(* CODESYS project SECoP-PLC
   Author: Zeus Castillo
   Company: ILL
   DefaultNamespace: SECoP
   Description: Library for configuring a Codesys-based PLC as a SEC Node
   DocFormat: reStructuredText
   LanguageModelAttribute: qualified-access-only
   Placeholder: SECoP
   Title: SECoP
   Version: 1.1.0.0

Project tree, tasks and I/O mapping:
  libraries: CAA Types Extern, 3.5.17.0 (CAA Technical Workgroup); CAA FB Factory, 3.5.19.0 (CAA Technical Workgroup); Common Behaviour Model, 4.0.0.0 (CODESYS); StringUtils, 3.5.20.0 (System); Util, 3.5.21.0 (System); Standard, 3.5.18.0 (System); SysMem, 3.5.17.0 (System); TcpUdpCommunication, 2.3.2.0 (Schneider Electric); JSON Utilities SL, 1.11.0.0 (CODESYS)
  global variables GCL
  global variables GPL
  global variables GVL
  data type ET_TimestampSource
  function block FB_SecNode [ST]: M_ReturnSecNodeError
  data type ST_SecNode
  data type ST_Timestamp
  program Server [ST]: A_MessageFragmentation, A_ParseClientMessage, A_ProcessClientRequest
  function GetLibVersion [ST]
  function GetLibVersionNumber [ST]
  function IsLibReleased [ST]
  data type ET_BaseClass
  data type ET_StatusCode
  function block FB_BaseModuleReadable [ST]: A_GenerateStatusDataReport, A_HandlePollintervalChange, A_ReturnErrorNoSuchCommand, A_ReturnErrorReadOnly, A_ReturnErrorWrongType, M_AddDataReportToReplyMessage, M_CheckIfDataIsNumeric, M_ExtractTargetLimitsFromTuple, M_GenerateTargetLimitsDataReport, M_JsonDecodeString, M_JsonEncodeString, M_ReturnRangeError
  data type ST_BaseModuleReadable
  data type ST_HandlePollinterval
  data type ST_ModuleStatus
  data type ST_Subscriber
  data type ST_TargetWrite
  data type ST_TargetDrive
  function block FB_diTargetDrive [ST]
  function block FB_IsStableNum [ST]
  function block FB_MonitorNumValue [ST]
  function block FB_MonitorSmallString [ST]
  function block FB_sTargetDrive [ST]
  global variables GPL_TcpServer_SE
*)

// ET_TimestampSource
{attribute 'qualified_only' := ''}
{attribute 'strict' := ''}
TYPE ET_TimestampSource :
(
	/// Value's timestamp to be obtained from the ECS (equipment that controls the hardware)
	Ecs := 1,
	/// Value's timestamp to be generated by this SEC node (this controller)				
	ThisSecNode := 2
);
END_TYPE

// ST_SecNode
TYPE ST_SecNode :
STRUCT
	// Firmware
	sFirmware: STRING := 'secnodeplc-1.0';
	// Protocol version
	sSecopVersion: STRING := 'V2019-09-16';	
	/// TCP server IP address
	sTcpServerIp: STRING(15);
	/// TCP server port
	uiTcpServerPort: UINT;
	// TCP server Eth interface link up
	xTcpServerInterfaceReady : BOOL:= FALSE;
	/// Default poll interval (to be used for modules that don´t have an independent pollinterval configured)
	timPollInterval: TIME := TIME#5S;
	/// Timestamp
	sTimestamp: STRING;
	/// Error report
	stErrorReport: ST_ErrorReport;
	// Module list
	asModule: ARRAY[1..GPL.Gc_uiMaxNoOfModules] OF STRING;
	// Action list
	asAction: ARRAY[1..GPL.Gc_uiMaxNoOfActions] OF STRING := ['*IDN?', 'describe', 'activate', 'deactivate', 'ping', 'read', 'change', 'do'];	
	// Structure report
	sStructureReport: STRING(GPL.Gc_uiMaxSizeMessage);
END_STRUCT
END_TYPE

// ST_Timestamp
TYPE ST_Timestamp :
STRUCT
	etSource: ET_TimestampSource;
	sValue: STRING;
END_STRUCT
END_TYPE

// ET_BaseClass
{attribute 'qualified_only' := ''}
{attribute 'strict' := ''}
TYPE ET_BaseClass : // Module's interface class 
(
	//Communicator := 0,
	Readable := 1,
	Writable := 2,
	Drivable := 3
);
END_TYPE

// ET_StatusCode
{attribute 'qualified_only' := ''}
{attribute 'strict' := ''}
TYPE ET_StatusCode : // Module's status code
(
	/// implemented
	Disabled := 0,
	Idle := 100,
	Warn := 200,
	Busy := 300,
	Error := 400,
	/// not implemented yet
	Persist := 101,
	Prepare := 301,
	Ramping := 302,
	Finish := 303
);
END_TYPE

// ST_BaseModuleReadable
TYPE ST_BaseModuleReadable :
STRUCT
	/// Interface class
	etInterfaceClass: ET_BaseClass;
	/// Name
	sName: STRING(80);
	/// Description
	sDescription: STRING(255);
	/// Current status of the module
	stStatus: ST_ModuleStatus;
	/// Polling interval of the module
	stPollInterval: ST_HandlePollinterval;
	/// Array of currently subscribed clients
	astSubscriberList: ARRAY[1..GPL.Gc_uiMaxNoOfClients] OF ST_Subscriber;
	/// Timestamp
	sTimestamp: STRING;
	/// Error report		
	stErrorReport: ST_ErrorReport;
END_STRUCT
END_TYPE

// ST_HandlePollinterval
TYPE ST_HandlePollinterval : // Module's poll intervall handling data
STRUCT
	lrValue: LREAL := 5.0;
	lrMin: LREAL := 0.5;
	lrMax: LREAL := 120.0;
	xReadOnly: BOOL := FALSE;
//	stPollintervalChangeClient: ST_Subscriber; // Client that sent the last pollinterval change request	
END_STRUCT
END_TYPE

// ST_ModuleStatus
TYPE ST_ModuleStatus : // Module's status data
STRUCT
	/// Staus code
	etCode: ET_StatusCode;
	/// Status description
	sDescription: STRING(GPL.Gc_uiMaxSizeDescription);
	/// Module inactive (flag) becomes unavailable for SECoP clients e.g. due to equipment configuration
	xInactive : BOOL; 
END_STRUCT
END_TYPE

// ST_Subscriber
TYPE ST_Subscriber : // Subscribed SECoP client data
STRUCT
	/// IP Address
	sIp: STRING(15);
	/// Assigned port number
	uiPort: UINT;
END_STRUCT
END_TYPE

// ST_TargetWrite
TYPE ST_TargetWrite : // Module's target change handling data
STRUCT
	/// Interlock
	xPossible: BOOL;
	/// Client that sent the last target change request	
	stTargetChangeClient: ST_Subscriber;
END_STRUCT
END_TYPE

// ST_TargetDrive
TYPE ST_TargetDrive : // Module's target drive handling data
STRUCT
	/// State machine. 0:Idle, 1:Request, 2:Applied in hardware, 3:Driving, 4:Completed
	uiState: UINT;
	/// Timeout to reach target
	timTimeout: TIME := TIME#10M0S0MS;
	/// Clients that sent a target change request while the target is still driving (module BUSY)
	astClientList: ARRAY[1..GPL.Gc_uiMaxNoOfClients] OF ST_Subscriber;
	/// Stay at current value command
	xStopCmd: BOOL;
	/// Client that sent the last stop command
	stStopCmdClient: ST_Subscriber;
END_STRUCT
END_TYPE

// GCL
{attribute 'qualified_only'}
VAR_GLOBAL CONSTANT
	Gc_uiMaxSizeIdentifier : UINT := 64; // Max. size of the specifier (e.g. module and accessible name) inside the message	
	Gc_uiMaxSizeAction : UINT := 64; // Max. size of action inside the message
	Gc_uiMaxSizeSpecifier : UINT := (GCL.Gc_uiMaxSizeIdentifier*2)+1; // Max. size of action inside the message
	Gc_uiMaxSizeClientMessage : UINT := Gc_uiMaxSizeAction+Gc_uiMaxSizeSpecifier+GPL.Gc_uiMaxSizeData+5; // Max. size of a messages received from SECoP clients	
	Gc_uiMaxNbOfSubmessages : UINT := 3; // Action, specier and data, separated by a white space character (\x20)
	Gc_dwLibVersionNumber : DWORD := 16777216; // Manual copy of GetLibVersionNumber(). Used in sec node app to create compile-time warning if > max.version supported by code generator
END_VAR

// GPL
{attribute 'qualified_only'}
{attribute 'parameterlist'}
VAR_GLOBAL CONSTANT
	Gc_uiMaxSizeMessage : UINT := 20000; // Max. size of a messages sent to SECoP clients
	Gc_uiMaxSizeData : UINT := 2000; // Max. size of the Data part of a SECoP message (a message = Action + Specifier (e.g. module:accessible) + Data)
	Gc_uiMaxSizeDescription : UINT := 500; // Max. size of the description in the Status or Error Report message 		
	Gc_uiMaxNoOfClients : UINT := 3; // Max. number of simultaneous connected clients
	Gc_uiMaxNoOfModules : UINT := 100; // Max. number of implemented modules in the SEC Node
	Gc_uiMaxNoOfActions : UINT := 15; // Max. number of implemented actions in the SEC Node
END_VAR

// GVL
{attribute 'qualified_only'}
VAR_GLOBAL
	G_st_SecNode : ST_SecNode; // SEC Node 
	G_ProcessModules : I_ProcessModules; // Process modules interface
	G_xProcessModulesAssigned : BOOL := FALSE; // (Flag) Process modules interface linked in application
	G_xJsonLibInstalled : BOOL := FALSE; // (Flag) JSON Utilities SL library installed in application (license required)
END_VAR

// GPL_TcpServer_SE
{attribute 'qualified_only'}
{attribute 'parameterlist'}
VAR_GLOBAL CONSTANT
	/// Max buffer size for sending/receiving data in one function call when using the Send/Receive methods from the TcpUdpCommunication library.
	/// M251: 2048. M262: 20000 for instance
	Gc_uiDataTransferChunkSize: UINT := 20000;
	/// Max. size of a message to be sent. If 'Gc_uiSendingMessageMaxSize' is greater than 'GVL_SaneTcp.Gc_uiDataTransferChunkSize', it will be split into several chunks that will be sent in consecutive function calls.
	/// For M262, it is recommended to be ser to same value as 'Gc_uiDataTransferChunkSize' to avoid splitting
	Gc_uiSendingMessageMaxSize: UINT := 20000;
END_VAR

// FB_SecNode
FUNCTION_BLOCK FB_SecNode
VAR_INPUT
	/// Action identifier (type of request: describe, activate...)
	i_sAction: STRING;
	/// Module name (empty for SEC node global actions which are not module-related)
	i_sModule: STRING(GCL.Gc_uiMaxSizeIdentifier);
	/// used as id for "ping" requests (the "pong" reply contains exactly the same id)	
	i_sArgument: STRING(((2 * GCL.Gc_uiMaxSizeIdentifier) + 1));
	/// Client sent a new request that needs processing
	i_xSyncModeRequest: BOOL;
	/// Action is implemented in this SEC node
	i_xActionIsImplemented: BOOL;
	/// Specifier format correct
	i_xSpecifierFormatOk: BOOL;
END_VAR
VAR_IN_OUT
	iq_stSecNode: ST_SecNode;
	/// Reply message
	iq_sReplyMessage: STRING(GPL.Gc_uiMaxSizeMessage);
END_VAR
VAR
	/// Flags
	iModuleIndex: INT;
END_VAR


// Process client request in sync mode
IF i_xSyncModeRequest THEN

	// Action not implemented
	IF NOT i_xActionIsImplemented THEN
		
		IF i_sAction='logging' OR i_sAction='check' THEN
			// Return "NotImplemented" error
			iq_stSecNode.stErrorReport.sClass := 'NotImplemented';
			iq_stSecNode.stErrorReport.sDescription := i_sAction;
			StrConcatA(pstFrom:= ADR(' is not implemented on this SEC node'), pstTo:= ADR(iq_stSecNode.stErrorReport.sDescription), iBufferSize:= UINT_TO_INT(GPL.Gc_uiMaxSizeDescription));
			M_ReturnSecNodeError(i_xErrorLatched:= FALSE);	
		
		ELSE // Return "ProtocolError" error
			iq_stSecNode.stErrorReport.sClass := 'ProtocolError';
			iq_stSecNode.stErrorReport.sDescription := 'Unknown action';
			M_ReturnSecNodeError(i_xErrorLatched:= FALSE);				
		END_IF

	// Specifier format error
	ELSIF NOT i_xSpecifierFormatOk THEN
		// Return "ProtocolError" error
		iq_stSecNode.stErrorReport.sClass := 'ProtocolError';
		iq_stSecNode.stErrorReport.sDescription := 'Specifier format error';
		M_ReturnSecNodeError(i_xErrorLatched:= FALSE);			
		
	ELSE
		
		// Process SEC Node request (global action which is not module-related)
		IF StrIsNullOrEmptyA(ADR(i_sModule)) = TRUE THEN
			// identification
				IF i_sAction = '*IDN?' THEN
					
					// Prepare reply message: ISSE,SECoP,(optional)<date indicating pre-release draft of the specin use>,< released version of SECoP>
					iq_sReplyMessage := 'ISSE,SECoP,2026-03-10,v2.0';
					M_AddTermToReplyMessage(i_etTerminator:= ET_Terminator.LineFeed); // Append line feed terminator to the message				
					
				// description
				ELSIF i_sAction = 'describe' THEN 
					
					// Prepare reply message: describing␣.␣<structure-report>
					iq_sReplyMessage := 'describing . ';
					StrConcatA(pstFrom:= ADR(iq_stSecNode.sStructureReport), pstTo:= ADR(iq_sReplyMessage), iBufferSize:= UINT_TO_INT(GPL.Gc_uiMaxSizeMessage));
					M_AddTermToReplyMessage(i_etTerminator:= ET_Terminator.LineFeed); // Append line feed terminator to the message	
				
				// activate updates
				ELSIF i_sAction = 'activate' THEN
		
					// Append action end message. Update messages were already inserted by the module FBs 			
					StrConcatA(pstFrom:= ADR('active'), pstTo:= ADR(iq_sReplyMessage), iBufferSize:= UINT_TO_INT(GPL.Gc_uiMaxSizeMessage));
					M_AddTermToReplyMessage(i_etTerminator:= ET_Terminator.LineFeed); // Append line feed terminator to the message				
	
				
				// deactivate updates
				ELSIF i_sAction = 'deactivate' THEN
					
					StrConcatA(pstFrom:= ADR('inactive'), pstTo:= ADR(iq_sReplyMessage), iBufferSize:= UINT_TO_INT(GPL.Gc_uiMaxSizeMessage));	
					M_AddTermToReplyMessage(i_etTerminator:= ET_Terminator.LineFeed); // Append line feed terminator to the message					
				
				// heartbeat. ping␣<identifier>
				ELSIF i_sAction = 'ping' THEN 
					
					// Prepare reply message: pong␣<identifier>␣<data-report>
					iq_sReplyMessage := 'pong ';
					StrConcatA(pstFrom:= ADR(i_sArgument), pstTo:= ADR(iq_sReplyMessage), iBufferSize:= UINT_TO_INT(GPL.Gc_uiMaxSizeMessage));
					StrConcatA(pstFrom:= ADR(' [null, {"t": '), pstTo:= ADR(iq_sReplyMessage), iBufferSize:= UINT_TO_INT(GPL.Gc_uiMaxSizeMessage));
					StrConcatA(pstFrom:= ADR(iq_stSecNode.sTimestamp), pstTo:= ADR(iq_sReplyMessage), iBufferSize:= UINT_TO_INT(GPL.Gc_uiMaxSizeMessage));
					StrConcatA(pstFrom:= ADR('}]'), pstTo:= ADR(iq_sReplyMessage), iBufferSize:= UINT_TO_INT(GPL.Gc_uiMaxSizeMessage));
					M_AddTermToReplyMessage(i_etTerminator:= ET_Terminator.LineFeed); // Append line feed terminator to the message
				END_IF
			
		ELSE // Check if the module specified on the client request is recognised. Return error otherwise
			FOR iModuleIndex := 1 TO UINT_TO_INT(GPL.Gc_uiMaxNoOfModules) BY 1 DO
				IF iq_stSecNode.asModule[iModuleIndex]=i_sModule THEN
					EXIT;
				END_IF
				IF StrIsNullOrEmptyA(ADR(iq_stSecNode.asModule[iModuleIndex])) THEN // end of module list reached
					// Return "NoSuchModule" error
					iq_stSecNode.stErrorReport.sClass := 'NoSuchModule';
					iq_stSecNode.stErrorReport.sDescription := i_sModule;
					StrConcatA(pstFrom:= ADR(' is not configured on this SEC node'), pstTo:= ADR(iq_stSecNode.stErrorReport.sDescription), iBufferSize:= UINT_TO_INT(GPL.Gc_uiMaxSizeDescription));
					M_ReturnSecNodeError(i_xErrorLatched:= FALSE);	
					EXIT;
				END_IF
			END_FOR				
		END_IF
	END_IF
END_IF

METHOD M_ReturnSecNodeError : BOOL
VAR_INPUT
	i_xErrorLatched: BOOL;
END_VAR

// Raise error flag
iq_stSecNode.stErrorReport.xActive := TRUE;	

// Build error report
StrConcatA(pstFrom:= ADR('error_'), pstTo:= ADR(iq_sReplyMessage), iBufferSize:= UINT_TO_INT(GPL.Gc_uiMaxSizeMessage));
StrConcatA(pstFrom:= ADR(i_sAction), pstTo:= ADR(iq_sReplyMessage), iBufferSize:= UINT_TO_INT(GPL.Gc_uiMaxSizeMessage));
StrConcatA(pstFrom:= ADR(' ["'), pstTo:= ADR(iq_sReplyMessage), iBufferSize:= UINT_TO_INT(GPL.Gc_uiMaxSizeMessage));	
StrConcatA(pstFrom:= ADR(iq_stSecNode.stErrorReport.sClass), pstTo:= ADR(iq_sReplyMessage), iBufferSize:= UINT_TO_INT(GPL.Gc_uiMaxSizeMessage));
StrConcatA(pstFrom:= ADR('","'), pstTo:= ADR(iq_sReplyMessage), iBufferSize:= UINT_TO_INT(GPL.Gc_uiMaxSizeMessage));
StrConcatA(pstFrom:= ADR(iq_stSecNode.stErrorReport.sDescription), pstTo:= ADR(iq_sReplyMessage), iBufferSize:= UINT_TO_INT(GPL.Gc_uiMaxSizeMessage));
StrConcatA(pstFrom:= ADR('",{"t":'), pstTo:= ADR(iq_sReplyMessage), iBufferSize:= UINT_TO_INT(GPL.Gc_uiMaxSizeMessage));
StrConcatA(pstFrom:= ADR(iq_stSecNode.sTimestamp), pstTo:= ADR(iq_sReplyMessage), iBufferSize:= UINT_TO_INT(GPL.Gc_uiMaxSizeMessage));
StrConcatA(pstFrom:= ADR('}]'), pstTo:= ADR(iq_sReplyMessage), iBufferSize:= UINT_TO_INT(GPL.Gc_uiMaxSizeMessage));	

// Append line feed terminator to the message
M_AddTermToReplyMessage(i_etTerminator:= ET_Terminator.LineFeed);	

// Unlatch error
IF NOT i_xErrorLatched THEN
	iq_stSecNode.stErrorReport.xActive := FALSE;
END_IF
END_METHOD

END_FUNCTION_BLOCK

// Server
PROGRAM Server // Sec node TCP server
VAR_INPUT
	xCmdClearResult: BOOL; /// Reset Cmd. Clear last diagnostic messages and alarms on rising edge
	xCmdDisconnectAll: BOOL; /// Disconnect all clients on rising edge	
	xCmdClose: BOOL; /// Stop listening (close port) on rising edge
END_VAR
VAR
{IF project_defined(SCHNEIDER_ELECTRIC)} 
	// SCHNEIDER_ELECTRIC Tcp Server handling
	fbTcpServer: FB_ASCIIoverTCPserver_SE;	
	fbReceivedData: ARRAY[1..TCPUDP.GPL.Gc_uiTCPServerMaxConnections] OF FB_MonitorNumValue;
	fbDisconnectedClientIp: ARRAY[1..TCPUDP.GPL.Gc_uiTCPServerMaxConnections] OF FB_MonitorSmallString;
	fbDisconnectedClientPort: ARRAY[1..TCPUDP.GPL.Gc_uiTCPServerMaxConnections] OF FB_MonitorNumValue;
	astClientInfo: ARRAY [1..TCPUDP.GPL.Gc_uiTCPServerMaxConnections] OF ST_ClientInfo_SE;
	asMessageToSend: ARRAY[1..TCPUDP.GPL.Gc_uiTCPServerMaxConnections] OF STRING(GPL_TcpServer_SE.Gc_uiSendingMessageMaxSize);
	sTcpServerState: STRING;
	sTcpServerResult: STRING;
	sLastErrorDiagMessage: STRING;
	uiNbOfConnectedClients: UINT;
	xPortOpen: BOOL;
	sDiagMessage: STRING;
	/// Auxiliary variables
	xMessageFragNeeded : BOOL := GPL_TcpServer_SE.Gc_uiDataTransferChunkSize < GPL_TcpServer_SE.Gc_uiSendingMessageMaxSize; // Message fragmentation needed	
	iStartPos: INT;
	iEndPos: INT;
	sDisconnectedCientIp: STRING;
	uiDisconnectedCientPort: UINT;
{END_IF}

	// Tcp Server handling
	// -----------------------
	uiClientId: UINT;
	fbBlink2s : BLINK;
	fbRtrig2s : R_TRIG;	
	xOnEvery2s : BOOL;
	x2sSinceStartup : BOOL := FALSE;
	xError: BOOL;
	xClientDisconnectedFlag: BOOL;
	xSyncModeRequest: BOOL;	
	stClientMonitored : ST_Subscriber;
	stClientDisconnected : ST_Subscriber;
	xFirstSecopClient: BOOL;
	xAllSecopClientsDone: BOOL;
	
	// Client request handling
	// -----------------------
	// Message to parse
	sMessageToParse: STRING(GCL.Gc_uiMaxSizeClientMessage);	
	// Action
	sAction: STRING(GCL.Gc_uiMaxSizeAction);
	// Specifier. Usually contains a module name and an accessible (parameter, property or command)
	sSpecifier: STRING(GCL.Gc_uiMaxSizeSpecifier);
	// Data
	sData: STRING(GPL.Gc_uiMaxSizeData);
	// Module
	sModuleName: STRING(GCL.Gc_uiMaxSizeIdentifier);
	// Accessible (parameter, a property or a command)
	sAccessibleName: STRING(GCL.Gc_uiMaxSizeIdentifier);
	/// Reply message
	sReplyMessage: STRING(GPL.Gc_uiMaxSizeMessage);
	/// Processs SEC node and module-wise requests
	fbSecNode: FB_SecNode;	
	/// Auxiliary variables
	iIndexSubMessage: INT;
	iCountSubMessages: INT;
	xActionIsImplemented: BOOL;
	xSpecifierFormatOk: BOOL;	
	iIndexAction: INT;
	etDelimiter: ET_Delimiter;
	etTerminator: ET_Terminator;
	iPos: INT;
	sTemp: STRING(GCL.Gc_uiMaxSizeClientMessage);	
END_VAR


// TCP server reset clock. If an exchange error occured, check 'q_sLastDiagMessage' for information on the last registered error 
fbBlink2s(ENABLE:= TRUE, TIMELOW:= T#1S, TIMEHIGH:= T#1S);
fbRtrig2s(CLK:= fbBlink2s.OUT);
xOnEvery2s := fbRtrig2s.Q;
IF xOnEvery2s THEN x2sSinceStartup:= TRUE; END_IF
xCmdClearResult := xError AND xOnEvery2s;

// Dispatcher. Prepare messages to be sent to clients
FOR uiClientId := 1 TO TCPUDP.GPL.Gc_uiTCPServerMaxConnections DO
	
	// Monitor disconnected clients
	{IF project_defined(SCHNEIDER_ELECTRIC)} 
	fbDisconnectedClientIp[uiClientId](i_sVar:= astClientInfo[uiClientId].sIp);
	fbDisconnectedClientPort[uiClientId](i_rVar:= UINT_TO_REAL(astClientInfo[uiClientId].uiPort));
	xClientDisconnectedFlag := 
		fbDisconnectedClientIp[uiClientId].q_xHasChanged AND fbDisconnectedClientIp[uiClientId].i_sVar ='' AND fbDisconnectedClientIp[uiClientId].q_sPreviousValue <> ''
		AND fbDisconnectedClientPort[uiClientId].q_xHasChanged 	AND fbDisconnectedClientPort[uiClientId].i_rVar <=0 AND fbDisconnectedClientPort[uiClientId].q_rPreviousValue > 0;
	IF xClientDisconnectedFlag THEN
		sDisconnectedCientIp :=  fbDisconnectedClientIp[uiClientId].q_sPreviousValue;
		uiDisconnectedCientPort :=  REAL_TO_UINT(fbDisconnectedClientPort[uiClientId].q_rPreviousValue);
		astClientInfo[uiClientId].stDataToSend.sData:='';
	END_IF
	{END_IF}
	
	// Detect new data from clients
	{IF project_defined(SCHNEIDER_ELECTRIC)} 
	fbReceivedData[uiClientId](i_rVar:= ULINT_TO_REAL(astClientInfo[uiClientId].uliTotalBytesReceived));	
	
	// Clear message buffer if the client is no longer connected when message fragmentation is used
	IF xMessageFragNeeded AND asMessageToSend[uiClientId] <> '' AND astClientInfo[uiClientId].uiPort<=0 THEN
		asMessageToSend[uiClientId]:='';
	END_IF
	{END_IF}	
		
	// Raise synchronous mode flag if there is a new client request to process
	{IF project_defined(SCHNEIDER_ELECTRIC)} 
	xSyncModeRequest := fbReceivedData[uiClientId].q_xHasChanged
						AND astClientInfo[uiClientId].stDataReceived.sData <> 'RN'
						AND astClientInfo[uiClientId].uiPort>0;
	{END_IF}
	
	// Parse client message in synchronous mode. Retrieve action, specifier (module & accessible) and data while looking for errors
	{IF project_defined(SCHNEIDER_ELECTRIC)} 	
	IF xSyncModeRequest THEN
		sMessageToParse:=astClientInfo[uiClientId].stDataReceived.sData;
		A_ParseClientMessage();
	END_IF
	{END_IF}	
	
	// Process client request (action) both in synchronous and asynchronous mode
	{IF project_defined(SCHNEIDER_ELECTRIC)} 
	stClientMonitored.sIp := astClientInfo[Server.uiClientId].sIp;
	stClientMonitored.uiPort := astClientInfo[Server.uiClientId].uiPort;
	stClientDisconnected.sIp := sDisconnectedCientIp;
	stClientDisconnected.uiPort := uiDisconnectedCientPort;
	xFirstSecopClient := uiClientId = 1;
	xAllSecopClientsDone := uiClientId = GPL.Gc_uiMaxNoOfClients;
	{END_IF} 		
	A_ProcessClientRequest();
	
	// Send message to client if there is data to send (push)
	{IF project_defined(SCHNEIDER_ELECTRIC)} 
	IF xMessageFragNeeded THEN // e.g. when using an M251 and message size > tcp buffer size (2048 bytes)
		Stu.StrConcatA(ADR(sReplyMessage), ADR(asMessageToSend[uiClientId]), UINT_TO_INT(SIZEOF(asMessageToSend[uiClientId])));
		IF asMessageToSend[uiClientId] <> '' THEN
			A_MessageFragmentation();
		END_IF
	ELSE 
		astClientInfo[uiClientId].stDataToSend.sData := sReplyMessage;
		IF astClientInfo[uiClientId].stDataToSend.sData <> '' THEN
			astClientInfo[uiClientId].axPushData := TRUE;
		END_IF
	END_IF
	{END_IF}

END_FOR;
	
// TCP Server accepting sockets from multiple clients
{IF project_defined(SCHNEIDER_ELECTRIC)} 
fbTcpServer(
	i_xEnable := x2sSinceStartup,
	i_xEthIfReady := GVL.G_st_SecNode.xTcpServerInterfaceReady,
	i_xCmdListen:= x2sSinceStartup AND GVL.G_st_SecNode.xTcpServerInterfaceReady,
	i_xCmdClose:= xCmdClose,
	i_xCmdDisconnectAll:= xCmdDisconnectAll, 
	i_xCmdClearResult:= xCmdClearResult, 
	i_sIpAddrServer:= GVL.G_st_SecNode.sTcpServerIp,
	i_uiTcpServerPort:= GVL.G_st_SecNode.uiTcpServerPort,
	i_timTimeoutInactivity:= T#30M,
	i_xTlsSelected:= FALSE,
	i_etCertVerifyMode:= TCPUDP.ET_CertVerifyMode.NotVerified,
	iq_astClientInfo := astClientInfo,
  	//q_astDataReceived := ,	
	//q_astConnectedClients=> , 
	q_uiNbOfConnectedClients=> uiNbOfConnectedClients,
	q_xPortOpen=> xPortOpen,
	q_sDiagMessage=> sDiagMessage,
	q_xDiag=> xError,
	q_sTcpServerState=> sTcpServerState,
	q_sTcpServerResult=> sTcpServerResult,
	q_sLastErrorDiagMessage=> sLastErrorDiagMessage);	

(*	
{ELSIF project_defined(WAGO)}
	...
{ELSIF project_defined(ABB)}
	...
...
*)
{ELSE}
	{error 'No platform defined! Please include it in the list of global defines in the Compile oprtions of the project settings}
{END_IF}

// Reset rising-edge-execution commands
xCmdClearResult := FALSE;
xCmdDisconnectAll := FALSE;
xCmdClose := FALSE;

ACTION A_MessageFragmentation:

{IF project_defined(SCHNEIDER_ELECTRIC)} 
astClientInfo[uiClientId].axPushData := TRUE;
IF StrLenA(pstData:= ADR(asMessageToSend[uiClientId])) < SIZEOF(astClientInfo[uiClientId].stDataToSend.sData) THEN // message is smaller than the buffer size
	astClientInfo[uiClientId].stDataToSend.sData := asMessageToSend[uiClientId]; // send whole message
	asMessageToSend[uiClientId] := ''; // no more data to be sent
ELSE // message is bigger than the buffer size
	iStartPos := 1;
	iEndPos :=  UINT_TO_INT(GPL_TcpServer_SE.Gc_uiDataTransferChunkSize)+1;
	stu.StrMidA(pst := ADR(asMessageToSend[uiClientId]),
						uiInputBufferSize := SIZEOF(asMessageToSend[uiClientId]),
						iLength := iEndPos - iStartPos,
						iPosition := iStartPos,
						pstResult := ADR(astClientInfo[uiClientId].stDataToSend.sData),
						uiResultBufferSize := SIZEOF(astClientInfo[uiClientId].stDataToSend.sData));
	// update remaining message to be sent on next iteration
	stu.StrDeleteA(pby:= ADR(asMessageToSend[uiClientId]), iLength:= iEndPos - iStartPos, iPosition:= iStartPos);				
END_IF
{END_IF}
END_ACTION

ACTION A_ParseClientMessage:

(* This action requires the following variables (declared in the Server POU) to be configured first
	sMessageToParse: STRING(GPL.Gc_uiMaxSizeMessage)
*)

// Initialise variables
sAction := '';
sSpecifier := '';
sData := '';
sModuleName := '';
sAccessibleName := '';
iCountSubMessages := 0;
StrCpyA(pBuffer := ADR(sTemp), pStr := ADR(sMessageToParse), iBufferSize := SIZEOF(sTemp));
iIndexSubMessage := 1;

// Loop to find and extract submessages
WHILE StrIsNullOrEmptyA(ADR(sTemp)) = FALSE AND (iIndexSubMessage < GCL.Gc_uiMaxNbOfSubmessages) DO
	etDelimiter := ET_Delimiter.Space;
    iPos := StrFindA(pst1 := ADR(sTemp), pst2 := ADR(etDelimiter), uiSearchStart := 1);

    // If delimiter is not found, break loop
    IF iPos <= 0 THEN
        EXIT;
    END_IF;
	
	CASE iIndexSubMessage OF
		
		1: // Extract Action
		    StrMidA(pst := ADR(sTemp), uiInputBufferSize := SIZEOF(sTemp),
        		    iLength := iPos - 1, iPosition := 1,
            		pstResult := ADR(sAction), uiResultBufferSize := SIZEOF(sAction));
					
		2: // Extract Specifier
   			StrMidA(pst := ADR(sTemp), uiInputBufferSize := SIZEOF(sTemp),
            		iLength := iPos - 1, iPosition := 1,
            		pstResult := ADR(sSpecifier), uiResultBufferSize := SIZEOF(sSpecifier));
	END_CASE

    // Remove extracted substring from temporary variable
    StrMidA(pst := ADR(sTemp), uiInputBufferSize := SIZEOF(sTemp),
            iLength := DINT_TO_INT(StrLenA(ADR(sTemp))) - iPos, iPosition := iPos + 1,
            pstResult := ADR(sTemp), uiResultBufferSize := SIZEOF(sTemp));

    iIndexSubMessage := iIndexSubMessage + 1;
END_WHILE;

// After quitting the loop, process the last remaining substring
IF StrIsNullOrEmptyA(ADR(sTemp)) = FALSE AND (iIndexSubMessage <= GCL.Gc_uiMaxNbOfSubmessages) THEN

	// Remove message terminator first
	etTerminator := ET_Terminator.CarriageReturn; // carriage return
	iPos := StrFindA(pst1 := ADR(sTemp), pst2 := ADR(etTerminator), uiSearchStart := 1);
	IF iPos >0 THEN
    	StrMidA(pst := ADR(sTemp), uiInputBufferSize := SIZEOF(sTemp),
            iLength := iPos-1, iPosition := 1,
            pstResult := ADR(sTemp), uiResultBufferSize := SIZEOF(sTemp));
	END_IF
	etTerminator := ET_Terminator.LineFeed; // line feed
	iPos := StrFindA(pst1 := ADR(sTemp), pst2 := ADR(etTerminator), uiSearchStart := 1);
	IF iPos >0 THEN
    	StrMidA(pst := ADR(sTemp), uiInputBufferSize := SIZEOF(sTemp),
            iLength := iPos-1, iPosition := 1,
            pstResult := ADR(sTemp), uiResultBufferSize := SIZEOF(sTemp));
	END_IF
	
	CASE iIndexSubMessage OF
		1: 	// Extract Action
			StrCpyA(pBuffer := ADR(sAction), pStr := ADR(sTemp), iBufferSize := SIZEOF(sAction));
			
		2: 	// Extract Specifier
			StrCpyA(pBuffer := ADR(sSpecifier), pStr := ADR(sTemp), iBufferSize := SIZEOF(sSpecifier));
		
		3: 	// Extract Data
			StrCpyA(pBuffer := ADR(sData), pStr := ADR(sTemp), iBufferSize := SIZEOF(sData));
	END_CASE
 
    iCountSubMessages := iIndexSubMessage; // Include the last substring
ELSE
    iCountSubMessages := iIndexSubMessage - 1; // Last index not used
END_IF;

// Check if retrived Action is recognised in the protocol
xActionIsImplemented := FALSE;
FOR iIndexAction := 1 TO UINT_TO_INT(GPL.Gc_uiMaxNoOfActions) BY 1 DO
	IF sAction = GVL.G_st_SecNode.asAction[iIndexAction] THEN 
		xActionIsImplemented := TRUE; 
		EXIT;
	END_IF
END_FOR

// If the message contains an implemented action and a specifier:
// - retrieves module and accessible from specifier if it contains a colon delimiter
// - otherwise, retrieves module name if the action is activate or deactivate for a specific module
// - otherwise, the specifier will be used as an argument if the action is ping
// - othwerise, raise format error

xSpecifierFormatOk := TRUE;
IF xActionIsImplemented AND StrIsNullOrEmptyA(ADR(sSpecifier)) = FALSE THEN
	
	etDelimiter := ET_Delimiter.Colon;
    iPos := StrFindA(pst1 := ADR(sSpecifier), pst2 := ADR(etDelimiter), uiSearchStart := 1);
	IF iPos > 0 THEN 
		
		// Extract Module
		StrMidA(pst := ADR(sSpecifier), uiInputBufferSize := SIZEOF(sSpecifier),
        		    iLength := iPos - 1, iPosition := 1,
            		pstResult := ADR(sModuleName), uiResultBufferSize := SIZEOF(sModuleName));

		// Extract Accessible
    	StrMidA(pst := ADR(sSpecifier), uiInputBufferSize := SIZEOF(sSpecifier),
        	    	iLength := DINT_TO_INT(StrLenA(ADR(sSpecifier))) - iPos, iPosition := iPos + 1,
            		pstResult := ADR(sAccessibleName), uiResultBufferSize := SIZEOF(sAccessibleName));
	
	// Specifier contains just a module name (without accessible) if the action is "activate" or "deactivate"
	ELSIF iPos = 0 AND (sAction='activate' OR sAction='deactivate') THEN
		sModuleName:=sSpecifier;
		
	ELSIF sAction<>'ping' THEN
		
		xSpecifierFormatOk := FALSE; // Specifier format error
    END_IF;
END_IF
END_ACTION

ACTION A_ProcessClientRequest:

(* This action requires the following variables (declared in the Server POU) to be configured first
 	stClientMonitored : ST_Subscriber;
	stClientDisconnected : ST_Subscriber;
	xSyncModeRequest: BOOL;	
	xDisconnectedCient: BOOL;
*)

// Initialise variables
sReplyMessage := '';

// Process SEC Node modules
// ====================================================
IF GVL.G_xProcessModulesAssigned THEN
	GVL.G_ProcessModules.Run(
		 i_sAction              := sAction,
		 i_sModuleRequested          := sModuleName,
		 i_sAccessibleName      := sAccessibleName,
		 i_sData                := sData,
		 i_stClientMonitored    := stClientMonitored,
		 i_stClientDisconnected := stClientDisconnected,
		 i_xClientDisconnectedFlag := xClientDisconnectedFlag,
		 i_xSyncModeRequest     := xSyncModeRequest,
		 i_xFirstSecopClient    := xFirstSecopClient,
		 i_xAllSecopClientsDone := xAllSecopClientsDone,
		 iq_sReplyMessage       := sReplyMessage);
END_IF

// Process SEC Node request (global action which is not module-related)
// ====================================================
fbSecNode(i_sAction:= sAction, 
			i_sModule:= sModuleName, 
			i_sArgument:= sSpecifier,
			i_xSyncModeRequest := xSyncModeRequest,
			i_xActionIsImplemented := xActionIsImplemented,
			i_xSpecifierFormatOk := xSpecifierFormatOk,
			iq_stSecNode:= GVL.G_st_SecNode,
			iq_sReplyMessage:= sReplyMessage);
END_ACTION

END_PROGRAM

// FB_MonitorNumValue
FUNCTION_BLOCK PUBLIC FB_MonitorNumValue // Detects when a numeric variable changes its value. Returns a rising edge plus the previous value
VAR_INPUT
	i_rVar 			:REAL;		// Numeric variable to monitor
END_VAR
VAR_OUTPUT
	q_xHasChanged 	:BOOL;		// Value has changed (Rising Edge)
	q_rPreviousValue:REAL;		// Previous value
END_VAR
VAR
	xInit			:BOOL := TRUE;
	rVarPrevious 	:REAL;
END_VAR


IF xInit THEN
	xInit := FALSE;
	rVarPrevious := i_rVar;
END_IF

q_xHasChanged := i_rVar <> rVarPrevious;

q_rPreviousValue := rVarPrevious;

rVarPrevious := i_rVar;

END_FUNCTION_BLOCK

// FB_MonitorSmallString
FUNCTION_BLOCK PUBLIC FB_MonitorSmallString
VAR_INPUT
	/// String variable to monitor, up to 255 char
	i_sVar: STRING(255);
END_VAR
VAR_OUTPUT
	/// Value has changed (Rising Edge)
	q_xHasChanged: BOOL;
	/// Previous value
	q_sPreviousValue: STRING(255);
END_VAR
VAR
	xInit: BOOL := TRUE;
	sVarPrevious: STRING;
END_VAR

IF xInit THEN
	xInit := FALSE;
	sVarPrevious := i_sVar;
END_IF

q_xHasChanged := i_sVar <> sVarPrevious;

q_sPreviousValue := sVarPrevious;

sVarPrevious := i_sVar;

END_FUNCTION_BLOCK

// GetLibVersion
// This function has been automatically generated from the project information.
FUNCTION GetLibVersion : VERSION
VAR_INPUT
	
END_VAR

GetLibVersion.uiMajor := 1;
GetLibVersion.uiMinor := 1;
GetLibVersion.uiServicePack := 0;
GetLibVersion.uiPatch := 0;

END_FUNCTION

// GetLibVersionNumber
// This function has been automatically generated from the project information.
FUNCTION GetLibVersionNumber : DWORD
VAR_INPUT
	
END_VAR

GetLibVersionNumber := 16842752;

END_FUNCTION

// IsLibReleased
// This function has been automatically generated from the project information.
FUNCTION IsLibReleased : BOOL
VAR_INPUT
	
END_VAR

IsLibReleased := TRUE;

END_FUNCTION

// FB_BaseModuleReadable
FUNCTION_BLOCK FB_BaseModuleReadable
VAR_INPUT
	// Action identifier (type of request: activate, read, change...)
	i_sAction: STRING(GCL.Gc_uiMaxSizeAction);
	// Module requested
	i_sModuleRequested: STRING(GCL.Gc_uiMaxSizeIdentifier);
	// Acessible (parameter, property or command)
	i_sAccessible: STRING(GCL.Gc_uiMaxSizeIdentifier);
	// Data
	i_sData: STRING(GPL.Gc_uiMaxSizeData);
	// Monitored client
	i_stClientMonitored: ST_Subscriber;
	// Disconnected client
	i_stClientDisconnected: ST_Subscriber;
	// (Flag) 'i_stClientDisconnected' just disconnected
	i_xClientDisconnectedFlag: BOOL;
	// (Flag) 'i_stClientMonitored' sent a new request that needs processing
	i_xSyncModeRequest: BOOL;
	// (Flag) 'i_stClientMonitored' is the first in server's list
	i_xFirstSecopClient: BOOL;
	// (Flag) All clients in server's list were processed	
	i_xAllSecopClientsDone: BOOL;
END_VAR
VAR_IN_OUT
	/// Reply message
	iq_sReplyMessage: STRING(GPL.Gc_uiMaxSizeMessage);
	// Module's name
	iq_sName: STRING(GCL.Gc_uiMaxSizeIdentifier);
	// Error report
	iq_stErrorReport: ST_ErrorReport;
	// Timestamo
	iq_sTimestamp: STRING;
	// Module status
	iq_stStatus: ST_ModuleStatus;
	// Polling interval
	iq_stPollInterval: ST_HandlePollinterval;
	// Subscriber list
	iq_astSubscriberList: ARRAY[1..GPL.Gc_uiMaxNoOfClients] OF ST_Subscriber;
END_VAR
VAR
	uiClientIndex: UINT;
	xClientFound: BOOL;
	xClientIsSubscribed: BOOL;
	sBuiltDataReport: STRING(GPL.Gc_uiMaxSizeData);
	lrPollintervalNewVal: LREAL;
	sStatusCode: STRING;
	sPollIntervalMin: STRING;
	sPollIntervalMax: STRING;
	xPollIntervalChanged: BOOL;
	sJsonStatusDescription: STRING(GPL.Gc_uiMaxSizeDescription*2);
	
    // JSON Utilities SL - Library handling
	// Encode
    factory    : JSON.JSONDataFactory;
    eErr       : FBF.ERROR;
    pJsonData  : POINTER TO JSON.JSONData;
    writer     : JSON.JSONByteArrayWriter;
    wsJsonData : WSTRING(GPL.Gc_uiMaxSizeDescription);
    wsRaw      : WSTRING(GPL.Gc_uiMaxSizeDescription);
    diLenW      : DINT;
	// Decode
	factoryDec    : JSON.JSONDataFactory;
	eErrDec       : FBF.ERROR;	
	pJsonDataDec  : POINTER TO JSON.JSONData;
	reader     : JSON.JSONByteArrayReader;
	stElement: JSON.JSONElement;
	wsJsonDec     : WSTRING(GPL.Gc_uiMaxSizeDescription);	
END_VAR

ACTION A_GenerateStatusDataReport:

sBuiltDataReport := '[';
sStatusCode := INT_TO_STRING(iq_stStatus.etCode);
StrConcatA(pstFrom:= ADR(sStatusCode), pstTo:= ADR(sBuiltDataReport), iBufferSize:= UINT_TO_INT(GPL.Gc_uiMaxSizeData));
StrConcatA(pstFrom:= ADR(','), pstTo:= ADR(sBuiltDataReport), iBufferSize:= UINT_TO_INT(GPL.Gc_uiMaxSizeData));
M_JsonEncodeString(i_sRawString:= iq_stStatus.sDescription, q_sJsonString=> sJsonStatusDescription);
StrConcatA(pstFrom:= ADR(sJsonStatusDescription), pstTo:= ADR(sBuiltDataReport), iBufferSize:= UINT_TO_INT(GPL.Gc_uiMaxSizeData));
StrConcatA(pstFrom:= ADR(']'), pstTo:= ADR(sBuiltDataReport), iBufferSize:= UINT_TO_INT(GPL.Gc_uiMaxSizeData));
END_ACTION

ACTION A_HandlePollintervalChange:

IF iq_stPollInterval.xReadOnly THEN // Configured as read-only
	
	// Return "ReadOnly" error	
	A_ReturnErrorReadOnly();	

ELSIF StrIsNullOrEmptyA(pstData:= ADR(i_sData)) THEN // No data to parse
	// Return "BadJSON" error
	A_ReturnErrorDataNotParsed();

ELSIF NOT M_CheckIfDataIsNumeric(i_sDataToParse:= i_sData, i_xMustBeInteger:= FALSE) THEN // Unexpected data type
	// Return "WrongType" error
	A_ReturnErrorWrongType();
	
ELSE // Process new value for pollinterval
	lrPollintervalNewVal := STRING_TO_LREAL(i_sData);
	IF lrPollintervalNewVal > iq_stPollInterval.lrMax OR lrPollintervalNewVal < iq_stPollInterval.lrMin THEN // Value out of range
		
		// Return "RangeError" error
		M_ReturnRangeError(i_RangeMin:= LREAL_TO_STRING(iq_stPollInterval.lrMin), i_RangeMax:= LREAL_TO_STRING(iq_stPollInterval.lrMax));
		
	ELSE	
		// Apply requested value
		iq_stPollInterval.lrValue := LIMIT(iq_stPollInterval.lrMin,lrPollintervalNewVal,iq_stPollInterval.lrMax);
		M_AddDataReportToReplyMessage(i_xReturnError := FALSE,  i_sAction := 'changed', i_sAccessible := i_sAccessible, i_sDataReport:= LREAL_TO_STRING(iq_stPollInterval.lrValue));
		xPollIntervalChanged := TRUE;
		// Register client that sent the pollinterval change request
		// iq_stPollInterval.stPollintervalChangeClient.sIp := i_stClientMonitored.sIp;
		// iq_stPollInterval.stPollintervalChangeClient.uiPort := i_stClientMonitored.uiPort;
	END_IF
END_IF
END_ACTION

ACTION A_ReturnErrorNoSuchCommand:

// Return "NoSuchCommand" error
iq_stErrorReport.sClass := 'NoSuchCommand';
iq_stErrorReport.sDescription := i_sAccessible;
StrConcatA(pstFrom:= ADR(' command is not implemented for module '), pstTo:= ADR(iq_stErrorReport.sDescription), iBufferSize:= UINT_TO_INT(GPL.Gc_uiMaxSizeDescription));			
StrConcatA(pstFrom:= ADR(i_sModuleRequested), pstTo:= ADR(iq_stErrorReport.sDescription), iBufferSize:= UINT_TO_INT(GPL.Gc_uiMaxSizeDescription));
M_ReplyWithErrorStraightAway(i_xErrorLatched:= FALSE);
END_ACTION

ACTION A_ReturnErrorReadOnly:

// Return "ReadOnly" error
iq_stErrorReport.sClass := 'ReadOnly';
iq_stErrorReport.sDescription := 'Parameter ';
StrConcatA(pstFrom:= ADR(iq_sName), pstTo:= ADR(iq_stErrorReport.sDescription), iBufferSize:= UINT_TO_INT(GPL.Gc_uiMaxSizeDescription));
StrConcatA(pstFrom:= ADR(':'), pstTo:= ADR(iq_stErrorReport.sDescription), iBufferSize:= UINT_TO_INT(GPL.Gc_uiMaxSizeDescription));
StrConcatA(pstFrom:= ADR(i_sAccessible), pstTo:= ADR(iq_stErrorReport.sDescription), iBufferSize:= UINT_TO_INT(GPL.Gc_uiMaxSizeDescription));
StrConcatA(pstFrom:= ADR(' can not be changed remotely'), pstTo:= ADR(iq_stErrorReport.sDescription), iBufferSize:= UINT_TO_INT(GPL.Gc_uiMaxSizeDescription));
M_ReplyWithErrorStraightAway(i_xErrorLatched:= FALSE);
END_ACTION

ACTION A_ReturnErrorWrongType:

// Return "WrongType" error
iq_stErrorReport.sClass := 'WrongType';
iq_stErrorReport.sDescription := i_sAction;
StrConcatA(pstFrom:= ADR(' '), pstTo:= ADR(iq_stErrorReport.sDescription), iBufferSize:= UINT_TO_INT(GPL.Gc_uiMaxSizeDescription));			
StrConcatA(pstFrom:= ADR(i_sModuleRequested), pstTo:= ADR(iq_stErrorReport.sDescription), iBufferSize:= UINT_TO_INT(GPL.Gc_uiMaxSizeDescription));			
StrConcatA(pstFrom:= ADR(':'), pstTo:= ADR(iq_stErrorReport.sDescription), iBufferSize:= UINT_TO_INT(GPL.Gc_uiMaxSizeDescription));			
StrConcatA(pstFrom:= ADR(i_sAccessible), pstTo:= ADR(iq_stErrorReport.sDescription), iBufferSize:= UINT_TO_INT(GPL.Gc_uiMaxSizeDescription));			
StrConcatA(pstFrom:= ADR(' can not be performed as the argument has the wrong type'), pstTo:= ADR(iq_stErrorReport.sDescription), iBufferSize:= UINT_TO_INT(GPL.Gc_uiMaxSizeDescription));			
M_ReplyWithErrorStraightAway(i_xErrorLatched:= FALSE);
END_ACTION

METHOD M_AddDataReportToReplyMessage : BOOL
VAR_INPUT
	/// Return error report in the message straight away IF SET TO true
	i_xReturnError: BOOL ;
	/// Action identifier (activate, read, change...)
	i_sAction: STRING;
	/// Accessible (parameter, property or command) name
	i_sAccessible: STRING(GCL.Gc_uiMaxSizeIdentifier);
	/// Data report
	i_sDataReport: STRING(GPL.Gc_uiMaxSizeData);
END_VAR
VAR
	sActionAux: STRING;
	xReturnErrorMessage: BOOL;
END_VAR

// Conditions for building an 'error_' message instead of a data report	
xReturnErrorMessage := 	i_xReturnError 
						OR (	i_sAccessible <> 'status'
								AND iq_stErrorReport.xActive 
								AND	(	(i_xSyncModeRequest AND (i_sAccessible = 'value' OR (i_sAccessible = 'target' AND i_sAction='change' )))
										OR (NOT i_xSyncModeRequest AND i_sAccessible = 'value')
									)		
							);
								
// Build data report
IF NOT xReturnErrorMessage THEN 

	// Action identifier to add in reply message
	IF i_sAction = 'activate' OR i_sAction = 'deactivate' OR i_sAction = 'change' OR i_sAction = 'update' THEN
		sActionAux := 'update ';
	ELSIF i_sAction = 'read' THEN
		sActionAux := 'reply ';
	ELSIF i_sAction = 'changed' THEN
		sActionAux := 'changed ';
	ELSIF i_sAction = 'check' THEN
		sActionAux := 'checked ';
	ELSIF i_sAction = 'do' THEN
		sActionAux := 'done ';
	ELSE
		sActionAux := i_sAction;
	END_IF
	
	// Update reply message
	StrConcatA(pstFrom:= ADR(sActionAux), pstTo:= ADR(iq_sReplyMessage), iBufferSize:= UINT_TO_INT(GPL.Gc_uiMaxSizeMessage));
	StrConcatA(pstFrom:= ADR(iq_sName), pstTo:= ADR(iq_sReplyMessage), iBufferSize:= UINT_TO_INT(GPL.Gc_uiMaxSizeMessage));	
	StrConcatA(pstFrom:= ADR(':'), pstTo:= ADR(iq_sReplyMessage), iBufferSize:= UINT_TO_INT(GPL.Gc_uiMaxSizeMessage));	
	StrConcatA(pstFrom:= ADR(i_sAccessible), pstTo:= ADR(iq_sReplyMessage), iBufferSize:= UINT_TO_INT(GPL.Gc_uiMaxSizeMessage));	
	StrConcatA(pstFrom:= ADR(' ['), pstTo:= ADR(iq_sReplyMessage), iBufferSize:= UINT_TO_INT(GPL.Gc_uiMaxSizeMessage));

	IF StrIsNullOrEmptyA(pstData:= ADR(i_sDataReport))=FALSE THEN
		StrConcatA(pstFrom:= ADR(i_sDataReport), pstTo:= ADR(iq_sReplyMessage), iBufferSize:= UINT_TO_INT(GPL.Gc_uiMaxSizeMessage));
	ELSE
		StrConcatA(pstFrom:= ADR('null'), pstTo:= ADR(iq_sReplyMessage), iBufferSize:= UINT_TO_INT(GPL.Gc_uiMaxSizeMessage));	
	END_IF

ELSE // Build error message

	// Action identifier to add in reply message
	IF i_sAction = 'activate' OR i_sAction = 'deactivate' THEN
		sActionAux := 'update';
	ELSE
		sActionAux := i_sAction;
	END_IF

	StrConcatA(pstFrom:= ADR('error_'), pstTo:= ADR(iq_sReplyMessage), iBufferSize:= UINT_TO_INT(GPL.Gc_uiMaxSizeMessage));
	StrConcatA(pstFrom:= ADR(sActionAux), pstTo:= ADR(iq_sReplyMessage), iBufferSize:= UINT_TO_INT(GPL.Gc_uiMaxSizeMessage));
	StrConcatA(pstFrom:= ADR(' '), pstTo:= ADR(iq_sReplyMessage), iBufferSize:= UINT_TO_INT(GPL.Gc_uiMaxSizeMessage));		
	StrConcatA(pstFrom:= ADR(iq_sName), pstTo:= ADR(iq_sReplyMessage), iBufferSize:= UINT_TO_INT(GPL.Gc_uiMaxSizeMessage));

	IF StrIsNullOrEmptyA(pstData:= ADR(i_sAccessible))=FALSE THEN
		StrConcatA(pstFrom:= ADR(':'), pstTo:= ADR(iq_sReplyMessage), iBufferSize:= UINT_TO_INT(GPL.Gc_uiMaxSizeMessage));	
		StrConcatA(pstFrom:= ADR(i_sAccessible), pstTo:= ADR(iq_sReplyMessage), iBufferSize:= UINT_TO_INT(GPL.Gc_uiMaxSizeMessage));
	END_IF

	StrConcatA(pstFrom:= ADR(' ["'), pstTo:= ADR(iq_sReplyMessage), iBufferSize:= UINT_TO_INT(GPL.Gc_uiMaxSizeMessage));	
	StrConcatA(pstFrom:= ADR(iq_stErrorReport.sClass), pstTo:= ADR(iq_sReplyMessage), iBufferSize:= UINT_TO_INT(GPL.Gc_uiMaxSizeMessage));
	StrConcatA(pstFrom:= ADR('","'), pstTo:= ADR(iq_sReplyMessage), iBufferSize:= UINT_TO_INT(GPL.Gc_uiMaxSizeMessage));
	StrConcatA(pstFrom:= ADR(iq_stErrorReport.sDescription), pstTo:= ADR(iq_sReplyMessage), iBufferSize:= UINT_TO_INT(GPL.Gc_uiMaxSizeMessage));
	StrConcatA(pstFrom:= ADR('"'), pstTo:= ADR(iq_sReplyMessage), iBufferSize:= UINT_TO_INT(GPL.Gc_uiMaxSizeMessage));	
END_IF

// Conclude message by appending the qualifier timestamp and a terminator
StrConcatA(pstFrom:= ADR(',{"t":'), pstTo:= ADR(iq_sReplyMessage), iBufferSize:= UINT_TO_INT(GPL.Gc_uiMaxSizeMessage));
StrConcatA(pstFrom:= ADR(iq_sTimestamp), pstTo:= ADR(iq_sReplyMessage), iBufferSize:= UINT_TO_INT(GPL.Gc_uiMaxSizeMessage));
StrConcatA(pstFrom:= ADR('}]'), pstTo:= ADR(iq_sReplyMessage), iBufferSize:= UINT_TO_INT(GPL.Gc_uiMaxSizeMessage));
M_AddTermToReplyMessage(i_etTerminator:= ET_Terminator.LineFeed); // Append line feed terminator to the message
END_METHOD

METHOD M_CheckIfDataIsNumeric : BOOL
VAR_INPUT
	/// Data to parse
	i_sDataToParse: STRING(GPL.Gc_uiMaxSizeData);
	/// TRUE => only integer allowed (no '.')	
	i_xMustBeInteger: BOOL;
END_VAR
VAR
	/// Working buffer and single-char temp (1 char + '\0')
	sWorkingString: STRING(GPL.Gc_uiMaxSizeData);
	sChar: STRING(2);
	/// Literals for comparisons
	sPlus: STRING(2) := '+';
	sMinus: STRING(2) := '-';
	sDot: STRING(2) := '.';
	sZero: STRING(2) := '0';
	sNine: STRING(2) := '9';
	/// Loop/state
	diLength: DINT;
	/// 1-based for StrMidA
	iPosition: INT;
	xHasDigit: BOOL;
	xHasDot: BOOL;
END_VAR

// Copy input and trim
sWorkingString := i_sDataToParse;
StrTrimA(pString:= ADR(sWorkingString));

// Empty -> not numeric
diLength := StrLenA(ADR(sWorkingString));
IF diLength = 0 THEN
    M_CheckIfDataIsNumeric := FALSE;
    RETURN;
END_IF;

// Optional leading sign at position 1
iPosition := 1;
StrMidA(
    pst                := ADR(sWorkingString),
    uiInputBufferSize  := SIZEOF(sWorkingString),
    iLength            := 1,
    iPosition          := iPosition,
    pstResult          := ADR(sChar),
    uiResultBufferSize := SIZEOF(sChar)
);
IF (StrCaseCmpA(ADR(sChar), ADR(sPlus)) = 0) OR
   (StrCaseCmpA(ADR(sChar), ADR(sMinus)) = 0) THEN
    iPosition := iPosition + 1;
    IF iPosition > diLength THEN
        // Sign alone is not a number
        M_CheckIfDataIsNumeric := FALSE;
        RETURN;
    END_IF;
END_IF;

// Scan characters from current position to end
WHILE iPosition <= diLength DO
    // sChar := substring(sWork, pos, 1)
    StrMidA(
        pst                := ADR(sWorkingString),
        uiInputBufferSize  := SIZEOF(sWorkingString),
        iLength            := 1,
        iPosition          := iPosition,
        pstResult          := ADR(sChar),
        uiResultBufferSize := SIZEOF(sChar)
    );

    // digit? ('0' <= sChar <= '9')
    IF (StrCaseCmpA(ADR(sChar), ADR(sZero)) >= 0) AND
       (StrCaseCmpA(ADR(sChar), ADR(sNine)) <= 0) THEN
        xhasDigit := TRUE;

    // single '.' allowed unless it must be an integer
    ELSIF (StrCaseCmpA(ADR(sChar), ADR(sDot)) = 0) THEN
        IF i_xMustBeInteger OR xHasDot THEN
            M_CheckIfDataIsNumeric := FALSE; // second dot
            RETURN;
        END_IF;
        xHasDot := TRUE;

    ELSE
        // Any other char (space, comma, letters incl. e/E, etc.) -> not numeric
        M_CheckIfDataIsNumeric := FALSE;
        RETURN;
    END_IF;

    iPosition := iPosition + 1;
END_WHILE;

// Must include at least one digit
M_CheckIfDataIsNumeric := xhasDigit;
END_METHOD

METHOD M_ExtractTargetLimitsFromTuple : BOOL
(*  Parses a JSON array/tuple expected to hold a target_limits pair, e.g. "[10.0, 300.0]" or "[-12, 12]".
    Returns TRUE when the input is a valid JSON array (starts with '[', ends with ']') AND contains 2 top-level elements
    q_uiSize   : number of top-level elements found.
    q_sLimitMin: first  element string (trimmed), populated only when q_uiSize = 2.
    q_sLimitMax: second element string (trimmed), populated only when q_uiSize = 2.
    If q_uiSize <> 2, q_sLimitMin and q_sLimitMax are cleared to empty strings. *)
VAR_INPUT
    /// Data to parse (expected JSON array format, e.g. "[-12, 12]")
    i_sDataToParse : STRING(GPL.Gc_uiMaxSizeData);	
END_VAR
VAR_OUTPUT
    /// Number of elements found inside the brackets/parentheses
    q_uiSize    : UINT;
	/// target limit min
    q_sLimitMin : STRING;
	/// target limit max
    q_sLimitMax : STRING;
END_VAR
VAR
    sWorkingString     : STRING(GPL.Gc_uiMaxSizeData);
    sComma : STRING(1) := ',';
    sOpenBracket : STRING(1) := '['; // open bracket
    sCloseBracket : STRING(1) := ']'; // close bracket
    iStringLength : INT;
	iInnerLen : INT;
   	iFirstComma : INT;	
    iCommaPos : INT;
    uiFrom : UINT;
END_VAR

M_ExtractTargetLimitsFromTuple := FALSE;
q_uiSize    := 0;
q_sLimitMin := '';
q_sLimitMax := '';
sWorkingString := i_sDataToParse;

// Remove surrounding whitespace in-place
StrTrimStartA(ADR(sWorkingString));
StrTrimEndA(ADR(sWorkingString));

// Need at least '[' and ']' (2 chars)
iStringLength := DINT_TO_INT(StrLenA(ADR(sWorkingString)));
IF iStringLength < 2 THEN
    RETURN;
END_IF;

// First character must be '[' (position 1)
IF StrFindA(ADR(sWorkingString), ADR(sOpenBracket), 1) <> 1 THEN
    RETURN;
END_IF;

// Last character must be ']' (search from position iStringLength → only matches there)
IF StrFindA(ADR(sWorkingString), ADR(sCloseBracket), INT_TO_UINT(iStringLength)) <> iStringLength THEN
    RETURN;
END_IF;

// Remove ']' first (position iStringLength), then '[' (position 1)
StrDeleteA(pby := ADR(sWorkingString), iLength := 1, iPosition := iStringLength);
StrDeleteA(pby := ADR(sWorkingString), iLength := 1, iPosition := 1);

// Trim whitespace just inside the brackets
StrTrimStartA(ADR(sWorkingString));
StrTrimEndA(ADR(sWorkingString));

// Empty tuple '[]'
IF StrLenA(ADR(sWorkingString)) = 0 THEN
    q_uiSize := 0;
    RETURN;
END_IF;

// Inner string length after bracket removal and trim
iInnerLen := DINT_TO_INT(StrLenA(ADR(sWorkingString)));

// Find first comma position (needed later for element extraction)
iFirstComma := StrFindA(ADR(sWorkingString), ADR(sComma), 1);

// Count top-level commas; elements = commas + 1
q_uiSize := 1;
uiFrom := 1;
REPEAT
    iCommaPos := StrFindA(ADR(sWorkingString), ADR(sComma), uiFrom);
    IF iCommaPos > 0 THEN
        q_uiSize := q_uiSize + 1;
        uiFrom := INT_TO_UINT(iCommaPos) + 1;
    END_IF;
UNTIL iCommaPos <= 0 END_REPEAT;

// Extract the two elements only when exactly 2 are present
IF q_uiSize = 2 AND iFirstComma > 0 THEN

    // Element 1: copy inner string into q_sLimitMin, then delete comma and everything after
    q_sLimitMin := sWorkingString;
    StrDeleteA(pby := ADR(q_sLimitMin), iLength := iInnerLen - iFirstComma + 1, iPosition := iFirstComma);
    StrTrimA(ADR(q_sLimitMin));
	
    // Element 2: delete first element + comma from sWorkingString, then trim
    // iFirstComma chars from position 1 = "10.0," → leaves " 300.0"
    StrDeleteA(pby := ADR(sWorkingString), iLength := iFirstComma, iPosition := 1);
    StrTrimA(ADR(sWorkingString));
    q_sLimitMax := sWorkingString;
	
	M_ExtractTargetLimitsFromTuple := TRUE;
	
ELSE
    q_sLimitMin := '';
    q_sLimitMax := '';
END_IF;
END_METHOD

METHOD M_GenerateTargetLimitsDataReport : BOOL
VAR_INPUT
 i_sLimitsMin: STRING;
 i_sLimitsMax: STRING;	
END_VAR

sBuiltDataReport := '[';
StrConcatA(pstFrom:= ADR(i_sLimitsMin), pstTo:= ADR(sBuiltDataReport), iBufferSize:= UINT_TO_INT(GPL.Gc_uiMaxSizeData));
StrConcatA(pstFrom:= ADR(','), pstTo:= ADR(sBuiltDataReport), iBufferSize:= UINT_TO_INT(GPL.Gc_uiMaxSizeData));
StrConcatA(pstFrom:= ADR(i_sLimitsMax), pstTo:= ADR(sBuiltDataReport), iBufferSize:= UINT_TO_INT(GPL.Gc_uiMaxSizeData));
StrConcatA(pstFrom:= ADR(']'), pstTo:= ADR(sBuiltDataReport), iBufferSize:= UINT_TO_INT(GPL.Gc_uiMaxSizeData));
END_METHOD

METHOD M_JsonDecodeString : BOOL
VAR_INPUT
    /// JSON-encoded string to decode (e.g. "hello world" — with surrounding quotes)
    i_sJsonString : STRING(GPL.Gc_uiMaxSizeDescription);
END_VAR
VAR_OUTPUT
    /// Decoded raw PLC string
    q_sRawString : STRING(GPL.Gc_uiMaxSizeDescription);
END_VAR
VAR
	diSrc  : DINT;
	diDst  : DINT;
	pbSrc  : POINTER TO BYTE;
	pbDst  : POINTER TO BYTE;
	pbTmp  : POINTER TO BYTE;
	bChar  : BYTE;
	bNext  : BYTE;
	sTmp : STRING(GPL.Gc_uiMaxSizeDescription + 2);  // +2 for '[' and ']'
END_VAR

// Handle JSON deserialization, double quotes, and escape characters

q_sRawString := '';
M_JsonDecodeString := FALSE;

IF NOT GVL.G_xJsonLibInstalled THEN // Use String Utils library 

	diLenW := TO_DINT(StrLenA(ADR(i_sJsonString)));
	
	// Must start with " (16#22) and end with "
	pbSrc := ADR(i_sJsonString);
	pbDst := ADR(q_sRawString);
	
	pbTmp := pbSrc;           bChar := pbTmp^;  // first char
	IF bChar <> 16#22 THEN RETURN; END_IF
	pbTmp := pbSrc + TO_UDINT(diLenW - 1);   bChar := pbTmp^;  // last char
	IF bChar <> 16#22 THEN RETURN; END_IF
	
	// Iterate between quotes, unescape
	diSrc := 1;    // skip opening "
	diDst := 0;
	
	WHILE diSrc <= diLenW - 2 DO
		pbTmp := pbSrc + TO_UDINT(diSrc);
		bChar := pbTmp^;
	
		IF bChar = 16#5C AND diSrc + 1 <= diLenW - 2 THEN  // backslash
			pbTmp := pbSrc + TO_UDINT(diSrc + 1);
			bNext := pbTmp^;
			CASE bNext OF
				16#22: bChar := 16#22;  // \" -> "
				16#5C: bChar := 16#5C;  // \\ -> \
				16#6E: bChar := 16#0A;  // \n -> LF
				16#72: bChar := 16#0D;  // \r -> CR
				16#74: bChar := 16#09;  // \t -> TAB
			ELSE
				bChar := bNext;
			END_CASE
			diSrc := diSrc + 2;
		ELSE
			diSrc := diSrc + 1;
		END_IF
	
		pbTmp := pbDst + TO_UDINT(diDst);
		pbTmp^ := bChar;
		diDst := diDst + 1;
	END_WHILE
	
	// Null terminate
	pbTmp := pbDst + TO_UDINT(diDst);
	pbTmp^ := 0;
	
	M_JsonDecodeString := TRUE;

ELSE // Use JSON Utilities SL library (license required) 
	
	// Create dedicated JSONData for decode (independent from encode's pJsonData)
	IF pJsonDataDec = 0 THEN
		pJsonDataDec := factoryDec.Create(eError => eErrDec);
	END_IF
	IF (pJsonDataDec = 0) OR (eErrDec <> FBF.ERROR.NO_ERROR) THEN
		RETURN; // out of memory
	END_IF
	
	// Parse the incoming JSON string
	// Wrap in [ ] so the parser accepts it — library requires object/array at root
	pJsonDataDec^.Clear();
	sTmp := '[';
	StrConcatA(pstFrom := ADR(i_sJsonString), pstTo := ADR(sTmp), iBufferSize := UINT_TO_INT(SIZEOF(sTmp)));
	StrConcatA(pstFrom := ADR(']'), pstTo := ADR(sTmp), iBufferSize := UINT_TO_INT(SIZEOF(sTmp)));
	wsJsonDec := STRING_TO_WSTRING(sTmp);

	reader(
		xExecute                 := TRUE,
		xAsyncMode               := FALSE,
		xIgnoreValueStringLength := TRUE,
		pwData                   := ADR(wsJsonDec),
		jsonData                 := pJsonDataDec^
	);
	
	// Index 0 = array wrapper, index 1 = the string element inside
	eErrDec := pJsonDataDec^.GetElementByIndex(diIndex := 1, jsonElement => stElement);
	
	IF eErrDec = FBF.ERROR.NO_ERROR AND stElement.eType = JSON.JSONType.WSTRING_VALUE THEN
		q_sRawString := WSTRING_TO_STRING(stElement.value.wsValue);
		M_JsonDecodeString := TRUE;
	END_IF
	
	// Reset reader
	reader(xExecute := FALSE, jsonData := pJsonDataDec^);

END_IF
END_METHOD

METHOD M_JsonEncodeString : BOOL
VAR_INPUT
	/// Raw PLC string to be JSON-encoded
	i_sRawString: STRING(GPL.Gc_uiMaxSizeDescription);
END_VAR
VAR_OUTPUT
	/// JSON-encoded string
	q_sJsonString: STRING(GPL.Gc_uiMaxSizeDescription*2);
END_VAR
VAR
    pbSrc  : POINTER TO BYTE;
    pbDst  : POINTER TO BYTE;
    pbTmp  : POINTER TO BYTE;
    bChar  : BYTE;
    diLenW : DINT;
    diSrc  : DINT;
    diDst  : DINT;
END_VAR

// Handle JSON serialization, double quotes, and escape characters

q_sJsonString := '';
M_JsonEncodeString := FALSE;

IF NOT GVL.G_xJsonLibInstalled THEN // Use String Utils library 
	
	diLenW := TO_DINT(StrLenA(ADR(i_sRawString)));
	
	pbSrc := ADR(i_sRawString);
	pbDst := ADR(q_sJsonString);
	
	// Write opening "
	pbTmp  := pbDst;
	pbTmp^ := 16#22;
	diDst  := 1;
	
	diSrc := 0;
	WHILE diSrc <= diLenW - 1 DO
		pbTmp := pbSrc + TO_UDINT(diSrc);
		bChar := pbTmp^;
	
		// If the character needs escaping, write the leading \ and remap bChar
		IF bChar = 16#22 OR bChar = 16#5C OR bChar = 16#0A OR bChar = 16#0D OR bChar = 16#09 THEN
			pbTmp  := pbDst + TO_UDINT(diDst);
			pbTmp^ := 16#5C;   // backslash prefix
			diDst  := diDst + 1;
			CASE bChar OF
				16#22: bChar := 16#22;  // " -> \"
				16#5C: bChar := 16#5C;  // \ -> \\
				16#0A: bChar := 16#6E;  // LF  -> \n
				16#0D: bChar := 16#72;  // CR  -> \r
				16#09: bChar := 16#74;  // TAB -> \t
			END_CASE
		END_IF
	
		// Write character (plain copy or second byte of escape sequence)
		pbTmp  := pbDst + TO_UDINT(diDst);
		pbTmp^ := bChar;
	
		diSrc := diSrc + 1;
		diDst := diDst + 1;
	END_WHILE
	
	// Write closing "
	pbTmp  := pbDst + TO_UDINT(diDst);
	pbTmp^ := 16#22;
	diDst  := diDst + 1;
	
	// Null terminate
	pbTmp  := pbDst + TO_UDINT(diDst);
	pbTmp^ := 0;
	
	M_JsonEncodeString := TRUE;
	
ELSE // Use JSON Utilities SL library (license required) 
	
	// Create JSON structure in memory: root will be a JSON string (not an array)
	IF pJsonData = 0 THEN
		pJsonData := factory.Create(eError => eErr);
	END_IF
	IF (pJsonData = 0) OR (eErr <> FBF.ERROR.NO_ERROR) THEN
		RETURN; // out of memory
	END_IF;
	
	// Root = JSON string at index 0, parent = -1 (root)
	wsRaw := STRING_TO_WSTRING(i_sRawString);
	pJsonData^.SetString(wsValue := wsRaw, diIndex := 0, diParentIndex := -1);
	
	// Serialize synchronously to WSTRING (no BUSY)
	wsJsonData := ""; // clear output buffer
	writer(
		xExecute    := TRUE,
		xAsyncMode  := FALSE,             // synchronous: completes in this cycle
		wsLinebreak := "",
		pwData      := ADR(wsJsonData),
		udiSize     := SIZEOF(wsJsonData),
		jsonData    := pJsonData^
	);
	
	// Remove trailing ", " added by JSON writer
	diLenW := StrLenW(ADR(wsJsonData));  // length in wide characters
	IF diLenW > 2 THEN
		wsJsonData[diLenW - 2] := 0;  // Terminator in UTF-16
		q_sJsonString := WSTRING_TO_STRING(wsJsonData);
		M_JsonEncodeString := TRUE;
	ELSE
		// Fallback: empty JSON string literal
		q_sJsonString := '';
	END_IF
	
	// reset FB
	writer(xExecute := FALSE, jsonData := pJsonData^);

END_IF
END_METHOD

METHOD M_ReturnRangeError : BOOL
VAR_INPUT
	i_RangeMin : STRING;
	i_RangeMax : STRING;
END_VAR

// Return "RangeError" error
iq_stErrorReport.sClass := 'RangeError';
iq_stErrorReport.sDescription := 'Value must be between ';
StrConcatA(pstFrom:= ADR(i_RangeMin), pstTo:= ADR(iq_stErrorReport.sDescription), iBufferSize:= UINT_TO_INT(GPL.Gc_uiMaxSizeDescription));	
StrConcatA(pstFrom:= ADR(' and '), pstTo:= ADR(iq_stErrorReport.sDescription), iBufferSize:= UINT_TO_INT(GPL.Gc_uiMaxSizeDescription));	
StrConcatA(pstFrom:= ADR(i_RangeMax), pstTo:= ADR(iq_stErrorReport.sDescription), iBufferSize:= UINT_TO_INT(GPL.Gc_uiMaxSizeDescription));	
M_ReplyWithErrorStraightAway(i_xErrorLatched:= FALSE);
END_METHOD

END_FUNCTION_BLOCK

// FB_diTargetDrive
FUNCTION_BLOCK PUBLIC FB_diTargetDrive
VAR_INPUT
    // Enable signal: when TRUE, the monitoring process starts
    i_xEnable      : BOOL;

    // Process values
    i_diPv         : DINT;	// Process value
    i_diSp         : DINT;	// Setpoint

    // Parameters
    i_diTolerance  : DINT;	// Absolute tolerance (± value around SP)
    i_timTimeout   : TIME;	// Maximum time allowed to reach the setpoint
END_VAR
VAR_OUTPUT
    q_xDone 	    : BOOL; // TRUE once reached or failed
    q_xSpReached    : BOOL;	// TRUE if PV reaches setpoint within tolerance before timeout
    q_xSpFail       : BOOL;	// TRUE if timeout expires without reaching setpoint
END_VAR
VAR
    fbTimeout      : TON;    // Timeout timer
END_VAR


IF NOT i_xEnable THEN
    // Reset everything when disabled
    fbTimeout(IN := FALSE);
    q_xSpReached := FALSE;
    q_xSpFail    := FALSE;
    q_xDone  := FALSE;
ELSE
    // Start / keep the timeout timer running while not terminated
    fbTimeout(IN := NOT q_xDone, PT := i_timTimeout);

    // Check if PV is within absolute tolerance window
    IF (NOT q_xDone) AND (ABS(i_diPv - i_diSp) <= i_diTolerance) THEN
        q_xSpReached := TRUE;
        q_xSpFail    := FALSE;
        q_xDone  := TRUE;           // Terminate: success
    END_IF

    // Check if timeout has expired without success
    IF (NOT q_xDone) AND fbTimeout.Q THEN
        q_xSpReached := FALSE;
        q_xSpFail    := TRUE;
        q_xDone  := TRUE;           // Terminate: failure
    END_IF
END_IF

END_FUNCTION_BLOCK

// FB_IsStableNum
FUNCTION_BLOCK PUBLIC FB_IsStableNum
VAR_INPUT
	/// Numeric variable to monitor	
	i_rVar: REAL;
	/// Tolerance in absolut value
	i_rTolerance: REAL;
	/// Timeout	
	i_timTimeout: TIME;
END_VAR
VAR_OUTPUT
	/// Value is stable
	q_xIsStable: BOOL;
END_VAR
VAR
	xInit: BOOL := TRUE;
	rVarPrevious: REAL;
	fbTimeout: TON;
END_VAR


IF xInit THEN
	xInit := FALSE;
	rVarPrevious:=i_rVar+i_rTolerance;
END_IF

fbTimeout(IN:= ABS(i_rVar - rVarPrevious)<=i_rTolerance, PT:= i_timTimeout, Q=> q_xIsStable, ET=> );

IF NOT fbTimeout.IN THEN
	rVarPrevious := i_rVar;
END_IF

END_FUNCTION_BLOCK

// FB_sTargetDrive
FUNCTION_BLOCK PUBLIC FB_sTargetDrive
VAR_INPUT
    i_xEnable     : BOOL;
    i_pbPv        : POINTER TO BYTE;   // ADR(iq_sValue)
    i_pbSp        : POINTER TO BYTE;   // ADR(iq_sTarget)
    i_timTimeout  : TIME;
END_VAR
VAR_OUTPUT
    q_xDone       : BOOL;
    q_xSpReached  : BOOL;   // PV = SP antes del timeout
    q_xSpFail     : BOOL;   // timeout expirado sin llegar
END_VAR
VAR
    fbTimeout     : TON;
END_VAR


IF NOT i_xEnable THEN
    // Reset everything when disabled
    fbTimeout(IN := FALSE);
    q_xSpReached := FALSE;
    q_xSpFail    := FALSE;
    q_xDone  := FALSE;
ELSE
    // Start / keep the timeout timer running while not terminated
    fbTimeout(IN := NOT q_xDone, PT := i_timTimeout);

    // Check if PV is within absolute tolerance window
    IF (NOT q_xDone) AND StrCmpA(pby1:= i_pbPv, pby2:= i_pbSp) = 0 THEN
        q_xSpReached := TRUE;
        q_xSpFail    := FALSE;
        q_xDone  := TRUE;           // Terminate: success
    END_IF

    // Check if timeout has expired without success
    IF (NOT q_xDone) AND fbTimeout.Q THEN
        q_xSpReached := FALSE;
        q_xSpFail    := TRUE;
        q_xDone  := TRUE;           // Terminate: failure
    END_IF
END_IF

END_FUNCTION_BLOCK

// Run
METHOD Run : BOOL
VAR_INPUT
	// Action
	i_sAction: STRING;
	// Module requested
	i_sModuleRequested: STRING(GCL.Gc_uiMaxSizeIdentifier);
	// Accessible (parameter, property or command)
	i_sAccessibleName: STRING(GCL.Gc_uiMaxSizeIdentifier);
	// Data
	i_sData: STRING(GPL.Gc_uiMaxSizeMessage);	
	// Monitored client
	i_stClientMonitored: ST_Subscriber;
	// Disconnected client
	i_stClientDisconnected: ST_Subscriber;
	// (Flag) 'i_stClientDisconnected' just disconnected
	i_xClientDisconnectedFlag: BOOL;
	// (Flag) 'i_stClientMonitored' sent a new request that needs processing
	i_xSyncModeRequest: BOOL;
	// (Flag) 'i_stClientMonitored' is the first in server's list
	i_xFirstSecopClient: BOOL;
	// (Flag) All clients in server's list were processed
	i_xAllSecopClientsDone: BOOL;	
END_VAR
VAR_IN_OUT
	/// Reply message
	iq_sReplyMessage: STRING(GPL.Gc_uiMaxSizeMessage);
END_VAR
END_METHOD

// M_UpdateStatusWhenDriveDone
METHOD M_UpdateStatusWhenDriveDone : BOOL
VAR_INPUT
	i_xDone : BOOL;
	i_xSpReached : BOOL;
	i_xTimeOutElapsed : BOOL;		
END_VAR
VAR
	sTargetDriveTimeout: STRING;	
END_VAR
IF i_xDone THEN
	IF I_xSpReached THEN // Target reached on time
		iq_stStatus.etCode := ET_StatusCode.Idle;
		iq_stStatus.sDescription := 'IDLE';
		iq_stErrorReport.sClass := '';
		iq_stErrorReport.sDescription := '';	
	ELSIF I_xTimeOutElapsed THEN // Timeout elapsed. Target not reached on time. Build error report
		iq_stStatus.etCode := ET_StatusCode.Error;
		iq_stStatus.sDescription := 'Target value not reached on time';
		iq_stErrorReport.xActive := TRUE;
		iq_stErrorReport.sClass := 'TimeoutError';
		iq_stErrorReport.sDescription := 'Target change took longer than the maximum allowed time: ';
		sTargetDriveTimeout := REAL_TO_STRING(TIME_TO_REAL(iq_stTargetDrive.timTimeout)/1000);
		StrConcatA(pstFrom:= ADR(sTargetDriveTimeout), pstTo:= ADR(iq_stErrorReport.sDescription), iBufferSize:= UINT_TO_INT(GPL.Gc_uiMaxSizeDescription));
		StrConcatA(pstFrom:= ADR(' seconds'), pstTo:= ADR(iq_stErrorReport.sDescription), iBufferSize:= UINT_TO_INT(GPL.Gc_uiMaxSizeDescription));
	END_IF
	iq_stTargetDrive.uiState := 4;
END_IF
END_METHOD
